//==================================================================================================
//							Beckhoff Automation Poland
//									23.05.2018
//	Struktura zawierajaca I/O odpowiedniego bloku
//  v1.1	|| TC v 3.1.4022.16		|| - zmiana nazwy struktury usuniete CoE
//  v1.0	|| TC v 3.1.4022.16		|| - pierwsza wersja
//==================================================================================================
TYPE ST_FBSetPositionOffsetIO:
STRUCT
	bExecute						: BOOL;								// Rising edge executes cmd
	lrPosition						: LREAL;
	bRelative						: BOOL;
	eFeedback						: Tc2_MC2_Drive.E_PositionOffsetFeedback;
	eMemory							: Tc2_MC2_Drive.E_PositionOffsetMemory;
	bBusy							: BOOL;
	bError							: BOOL;
	udiErrorID						: UDINT;
	uiSecErrId						: UINT;								// Sercos Error ID for AX5000, CanOpen error ID for AX8000
END_STRUCT
END_TYPE

(* stored: Version 1.1.0.1, ProductVersion 3.1.4026.13, FileIdentifier a8b31f7a2d5612e7434ea3682a00361334c6cb53, FileSignature 8988246480ee1da608a7389464828cef80f96bde7424730204c72e951962fbf25993269370f266b6426dec7133fbf9782ce7270fcf87fc927717aed5860f9d71fa13825f948955134468bd83378c0e1543d212a76d276ed2dac06791924e1d7552b0117ff66b939872a4f38f47c860088741afeff80e7f6032a080afcaf26be1c39f8c0ba8c21d55639d4f94cac04e48ebceb8def51d82462ceb1451afa571402331cdb90013777ead86cd643c9e37b854fbaf876ecb39baf6bbf586b8bd868a3970215ff9504ba0fbb0f375061a8a94b8c372e9d41d61d14989ef0a2bd17e2f66b12b0ed835c0a30090d22a8562e22991d0afb8cfc79d8ab7e585aee8d8313e
   DUT ST_FBSetPositionOffsetIO: Id {490272c2-877f-494c-8bee-4cb06a7d96cd} *)
